TYPE E_CommandType :
(
    CMD_NONE                := 0,
    CMD_MODE_REQUEST        := 1,
    CMD_JOG_POSITIVE        := 2,
    CMD_JOG_NEGATIVE        := 3,
    CMD_MOVE_ABSOLUTE       := 4,
    CMD_MOVE_RELATIVE       := 5,
    CMD_MOVE_VELOCITY       := 6,
    CMD_STOP                := 7,
    CMD_RESET               := 8,
    CMD_HOME                := 9,
    CMD_ACK_ALARM           := 10,
    CMD_RESET_ALL_ALARMS    := 11
);
END_TYPE

(* stored: Version 1.1.0.1
   DUT E_CommandType: Id {25BC38EA-DFB4-4C5B-E142-E3724460142E} *)
